FUNCTION_BLOCK PUBLIC FB_PizzaItalianStyle IMPLEMENTS I_Pizza
VAR_INPUT
END_VAR
VAR_OUTPUT
END_VAR
VAR
END_VAR

METHOD PUBLIC GetPrice : LREAL
GetPrice := 4.5;
END_METHOD

END_FUNCTION_BLOCK

(* stored: Version 1.1.0.1, ProductVersion 3.1.4022.12
   POU FB_PizzaItalianStyle: Id {1c3477c4-341a-4dc9-b0e0-53d15dcbfd97}, SpecialFunc None
   Method GetPrice: Id {8ec69f28-78d1-4703-a427-86e7a5cbe010} *)
